RoboDK station: Assistive_UR5e_Maria.rdk

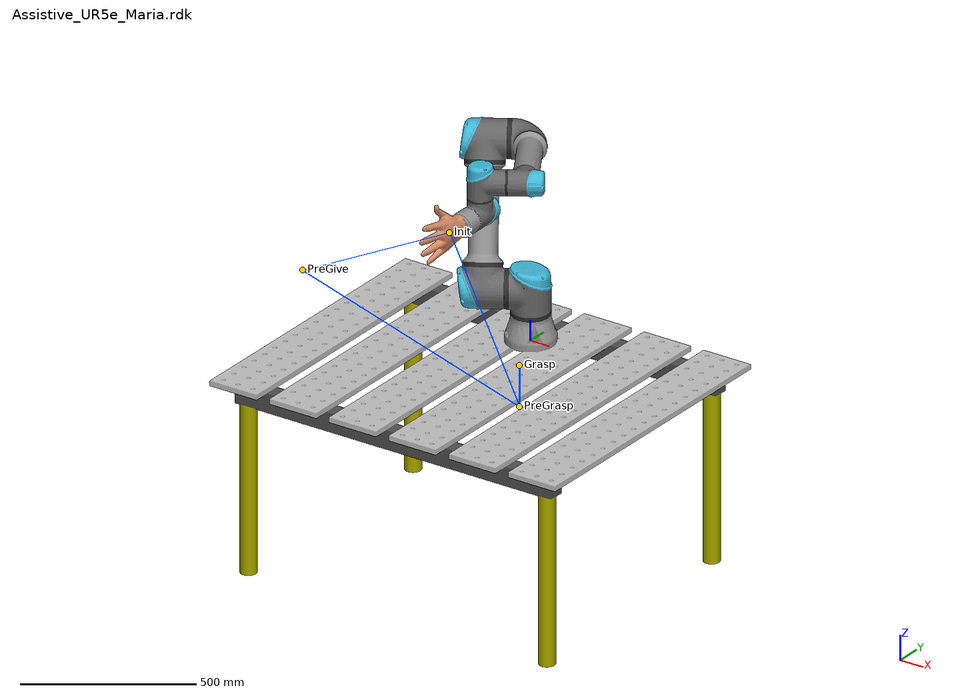
[picture v0: the station drawn from its stored meshes, robots at their saved joint values, targets as dots, program paths as lines]
Station Assistive_UR5e_Maria (saved by RoboDK 5.9.2). Poses are relative to the parent item; angles as X-Y-Z fixed-axis rotations.
  - frame UR5e Base at (0, 0, 0) mm
    - robot UR5e: 6 axes, payload 5 kg, reach 850 mm, repeatability 0.03 mm, weight 18.4 kg
        modified DH rows (alpha deg, a mm, theta deg, d mm): 0, 0, 0, 162.5; 90, 0, 180, 0; 0, 425, 0, 0; 0, 392.25, 0, 133.3; -90, 0, 0, 99.7; 90, 0, 180, 99.6
        joint limits [-360, -360, -360, -360, -360, -360] to [360, 360, 360, 360, 360, 360]; home [0, -90, -90, 0, 90, 0]; saved at [-57.836, -65.392, -107.167, 172.559, -57.836, 0]
      - tool Hand, TCP at (0, 0, 50) mm, size 54.8 x 155.9 x 193.5 mm, geometry from Hand.stl
  - frame World at (0, 0, 0) mm
    - object Table at (0, 0, 0) mm, size 1193.8 x 965.2 x 609.6 mm, geometry from welding_table.sld
    - target Init (Cartesian target) at (0, -400, 500) mm, rotated rx 90 ry 0 rz 0 deg; joints [-57.836, -65.392, -107.167, 172.559, -57.836, 0] of UR5e
    - target PreGrasp (Cartesian target) at (360.11, -569.97, 120.12) mm, rotated rx 54.52 ry 89.99 rz -35.48 deg; joints [-35.48, -127.85, -97.34, 225.2, -35.48, -90] of UR5e
    - target Grasp (Cartesian target) at (360.11, -569.97, 250.12) mm, rotated rx 55.48 ry 89.99 rz -34.52 deg; joints [-35.48, -117.221, -91.855, 209.086, -35.48, -90] of UR5e
    - target PreGive (Cartesian target) at (-389.89, -569.97, 340.12) mm, rotated rx 141.7 ry 89.99 rz -35.8 deg; joints [-100.541, -120.53, -72.544, 193.041, -13.041, -89.961] of UR5e
    - target Give (Cartesian target) at (-389.89, -569.97, 340.12) mm, rotated rx 179.99 ry 62.49 rz 2.49 deg; joints [-102.105, -135.503, -45.62, 116.965, -30.876, -29.428] of UR5e
  - program Init (3 instructions, listed below)
  - program Give (10 instructions, listed below)
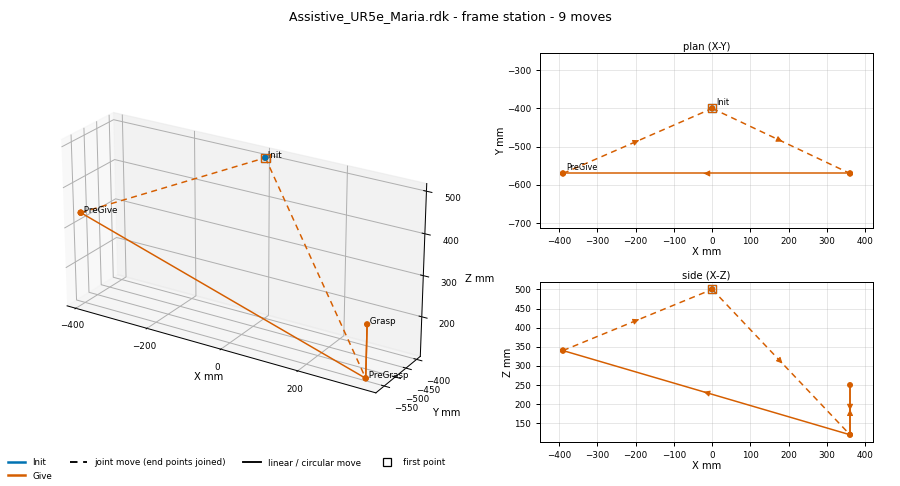
[picture p0: tool path of Assistive_UR5e_Maria.rdk in frame station, 9 of 9 moves have a stored position in this frame; points joined in program order, loops and branches not executed]

--- program Init (robot UR5e) ---
  Est. Ref.: UR5e Base
  Est. herr: Hand
  MoveJ (Init)

--- program Give (robot UR5e) ---
  Set Ref.: World
  Set Tool: Hand
  MoveJ (Init)
  MoveJ (PreGrasp)
  MoveL (Grasp)
  MoveL (PreGrasp)
  MoveL (PreGive)
  MoveL (Give)
  MoveL (PreGive)
  MoveJ (Init)
